FUNCTION_BLOCK QueueItem EXTENDS LinkedListItem IMPLEMENTS I_QueueItem
VAR
END_VAR

END_FUNCTION_BLOCK

(* stored: Version 1.1.0.1, ProductVersion 3.1.4024.12
   POU QueueItem: Id {698fcf05-9d43-4937-b564-68001b14eca1}, SpecialFunc None *)
